{attribute 'qualified_only'}
VAR_GLOBAL
	LaudaChillerWrites : ST_Chiller_Writes;
	LaudaChillerReads : ST_Chiller_Reads;
END_VAR

(* stored: Version 1.1.0.1
   GVL GVL_Lauda: Id {dfdd94c5-b704-49fd-92e0-b472372d4a00} *)
